PROGRAM Intfc_Left_PK
VAR
END_VAR

// NETWORK 1

END_PROGRAM

(* stored: Version 1.1.0.1, ProductVersion 3.1.4022.11
   POU Intfc_Left_PK: Id {2f559aba-41f8-4b56-8a63-c2206897e885}, SpecialFunc None *)
